// TIA Portal V19 export
TYPE "LAF_typeEnableControlInterfaces"
// Enable interfaces to control unit
// stored: Access Published
   STRUCT
      local : Bool;   // Enable local control interface
      hmi : Bool := true;   // Enable HMI control interface
      remote : Bool;   // Enable remote control interface
   END_STRUCT;
END_TYPE
